{attribute 'reflection'}
FUNCTION_BLOCK ABSTRACT HmiFunction EXTENDS CyclicComponent IMPLEMENTS I_HmiFunction
VAR
	{attribute 'instance-path'}
	{attribute 'noinit'}
	{attribute 'hide'}
	_InstancePath : STRING;
	{attribute 'hide'}
	_Enabled : BOOL := TRUE;
	{attribute 'hide'}
	_ControlType : STRING := 'Default';
	{attribute 'hide'}
	_LinkObject : STRING := 'DefaultFunction_HMI';
END_VAR

PROPERTY ABSTRACT ControlObject : I_Base
SET
END_SET
END_PROPERTY

{attribute 'monitoring' := 'call'}
PROPERTY ControlType : STRING
GET
ControlType := _ControlType;
END_GET
SET
_ControlType := ControlType;
END_SET
END_PROPERTY

METHOD CyclicLogic
END_METHOD

METHOD Disable
_Enabled := FALSE;
END_METHOD

METHOD Enable
_Enabled := TRUE;
END_METHOD

{attribute 'monitoring' := 'call'}
PROPERTY Enabled : BOOL
GET
Enabled := _Enabled;
END_GET
END_PROPERTY

{attribute 'monitoring' := 'call'}
PROPERTY InstancePath : STRING
GET
InstancePath := _InstancePath;
END_GET
END_PROPERTY

{attribute 'monitoring' := 'call'}
PROPERTY LinkObject : STRING
GET
LinkObject := _LinkObject;
END_GET
SET
_LinkObject := LinkObject;
END_SET
END_PROPERTY

END_FUNCTION_BLOCK

(* stored: Version 1.1.0.1, ProductVersion 3.1.4026.18
   POU HmiFunction: Id {697ccf64-b10d-4781-bd30-b5ead327a0b4}, SpecialFunc None
   Property ControlObject: Id {0f95bf7f-f01d-467e-849f-499a779aa19e}
   Set Set: Id {878878fb-8af4-4ea7-ac96-7bd7c21d2671}
   Property ControlType: Id {77ff7cd9-b54e-46ea-807a-e67282a6c5e7}
   Get Get: Id {45d21831-40a2-4864-9a31-569a10ed734b}
   Set Set: Id {20fb0eea-4e80-4678-a637-89ec0dbd058a}
   Method CyclicLogic: Id {19083ff2-6cba-40d5-b290-f0b910b9728c}
   Method Disable: Id {addc4d4a-52a1-4238-9d50-c8eb5d4a1fde}
   Method Enable: Id {861a72bc-57ae-4fe0-bd19-2190f2215cfd}
   Property Enabled: Id {180388bb-9c0d-48bf-a27a-840c862561d7}
   Get Get: Id {f6dc17ae-fcd8-4cde-9154-8a1e7d9caffb}
   Property InstancePath: Id {c2c255d6-ef36-445e-9c81-df65a7ec19d3}
   Get Get: Id {0c816d00-1eb8-4948-9590-6d0349356a86}
   Property LinkObject: Id {3ede90da-cffa-4f8e-82ce-df48fef853c2}
   Get Get: Id {d436a3ba-ddda-47a1-abf1-3698d08a9483}
   Set Set: Id {3e0964cb-1574-4398-bf96-ee63f0edaa16} *)
